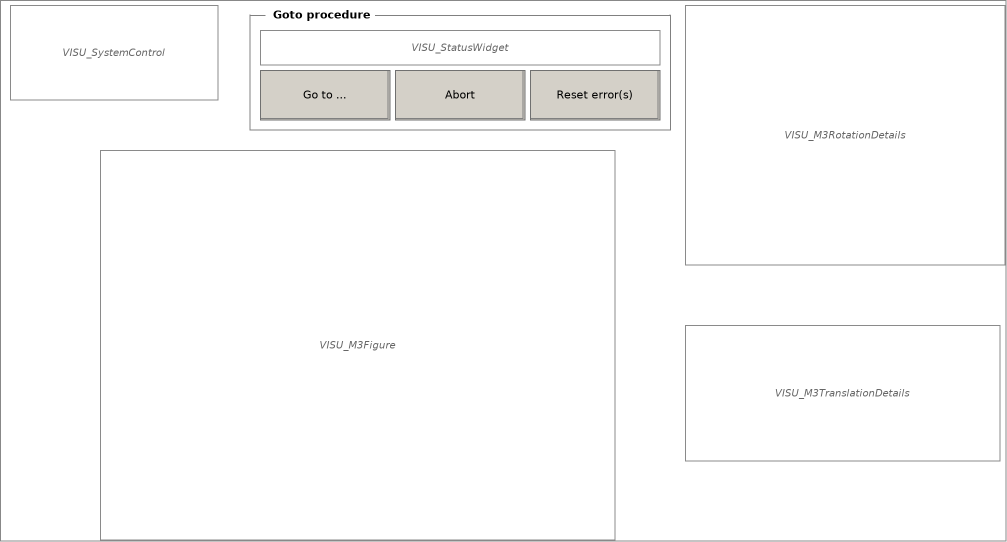
VISUALIZATION VISU_M3Overview  // 1007x542
VAR_IN_OUT
	m3 : M3;
    m3Widget : M3Widget;
END_VAR
    Frame (100,150 515x390)
        shows VISU_M3Figure(m3 := m3, widget := m3Widget, hideDetails := m3Widget.NO)
    Frame (685,5 320x260)
        shows VISU_M3RotationDetails(ref := m3.parts.rotation, widget := m3Widget.rotation)
    Button (260,70 130x50), "Go to ..."
        OnMouseClick: OpenDialog Dialog=VISU_M3TargetDialog, OpenModal=True, OpenCentered=True
    Frame (10,5 208x95)
        shows VISU_SystemControl(status := m3Widget.actualStatus, button_initialize := m3Widget.button_initialize, button_operating := m3Widget.button_operating, button_locking := m3Widget.button_locking)
    Frame (685,325 315x136)
        shows VISU_M3TranslationDetails(ref := m3.parts.translation)
    Frame (260,30 400x35)
        shows VISU_StatusWidget(widget := m3Widget.gotoProcedureStatus)
    Button (395,70 130x50), "Abort", input disabled if: m3.processes.abort.statuses.enabledStatus.disabled
        OnMouseClick: execute { m3.processes.abort.do_request := TRUE; }
    Button (530,70 130x50), "Reset error(s)", input disabled if: m3.processes.reset.statuses.enabledStatus.disabled
        OnMouseClick: execute { m3.processes.reset.do_request := TRUE; }
    Label (270,5 95x20), "Goto procedure"
    Polyline (375,15) (670,15) (670,130) (250,130) (250,15) (265,15)
END_VISUALIZATION

(* stored: Version 1.1.0.1, ProductVersion 3.1.4019.2
   Visu VISU_M3Overview: Id {4cbb2207-3d2c-406b-8519-d11eb0db6dd7} *)
